{attribute 'linkalways'} 
{attribute 'no_explicit_call' := 'This FB is a CLASS and must be accessed using methods or properties'}
{attribute 'enable_dynamic_creation'}
FUNCTION_BLOCK Node_F_VN_AppendToContainer_TcVnVector3_SINT EXTENDS VisionNode
VAR
    aElement : _TcVnVector3_SINT;
    ipContainer : _ITcVnContainer;
    hrPrev : _HRESULT(S_OK);
	hresult : _HRESULT(S_OK);
END_VAR

METHOD PUBLIC  Clone : I_Node
VAR
	pNode : POINTER TO Node_F_VN_AppendToContainer_TcVnVector3_SINT;
END_VAR
pNode := __NEW(Node_F_VN_AppendToContainer_TcVnVector3_SINT);
Clone := pNode^;
END_METHOD

METHOD FB_init : BOOL
VAR_INPUT
	bInitRetains : BOOL; // if TRUE, the retain variables are initialized (warm start / cold start)
	bInCopyCode : BOOL;  // if TRUE, the instance afterwards gets moved into the copy code (online change)
END_VAR
AddInput('aElement', aElement);
AddInput('ipContainer', ipContainer);
AddInput('hrPrev', hrPrev);
AddOutput('ipContainer', ipContainer);
AddOutput('hresult',hresult);
END_METHOD

METHOD PROTECTED OnExecute : HRESULT
hresult.Value := F_VN_AppendToContainer_TcVnVector3_SINT(
    aElement := aElement.Value,
	ipContainer := ipContainer.Value,
	hrPrev:= hrPrev.Value);
END_METHOD

METHOD PUBLIC PreExecutionCheck
VAR_INPUT
	Check : I_PreExecutionChecks;
END_VAR
Check.IsTrue(ipContainer.IsValid, 'ipContainer must be a valid container');
END_METHOD

END_FUNCTION_BLOCK

(* stored: Version 1.1.0.1, ProductVersion 3.1.4024.13
   POU Node_F_VN_AppendToContainer_TcVnVector3_SINT: Id {46f69f66-c1c7-4411-ae97-3dd51e946835}, SpecialFunc None
   Folder Constructor: Id {c126ac32-a7b3-404c-b67c-495ee321f321}
   Method Clone: Id {0b8a25c0-6e55-43d0-ade8-396038e769e5}
   Method FB_init: Id {692338f9-c965-4949-85f0-f09a7561d2b2}
   Method OnExecute: Id {539987c1-7878-42de-b713-60b1873ca4b6}
   Method PreExecutionCheck: Id {9c6c7e3b-2adc-4eef-bb59-4cad00c57014} *)
